FUNCTION_BLOCK FB_TelescopeAuxiliary
VAR
	tempSensorM1   		AT%I*: INT;
	tempSensorM1cell	AT%I*: INT;
	tempSensorM2   		AT%I*: INT;
	tempSensorFlange	AT%I*: INT;
	fbComm				: I_Comm;
END_VAR
VAR_OUTPUT
	tempM1				: REAL;
	tempM1cell			: REAL;
	tempM2				: REAL;
	tempFlange			: REAL;
END_VAR

tempM1 		:= tempSensorM1 / 32767.0 * 150.0 - 50.0; 
tempM1cell 	:= tempSensorM1cell / 32767.0 * 150.0 - 50.0;
tempM2 		:= tempSensorM2 / 32767.0 * 150.0 - 50.0;
tempFlange 	:= tempSensorFlange / 32767.0 * 150.0 - 50.0;

//FB_Init is always available implicitly and it is used primarily for initialization.
//The return value is not evaluated. For a specific influence, you can also declare the
//methods explicitly and provide additional code there with the standard initialization
//code. You can evaluate the return value.
METHOD FB_Init: BOOL
VAR_INPUT
    bInitRetains	: BOOL; // TRUE: the retain variables are initialized (reset warm / reset cold)
    bInCopyCode		: BOOL;  // TRUE: the instance will be copied to the copy code afterward (online change)
	comm			: I_Comm;	   
END_VAR
THIS^.fbComm := comm;
END_METHOD

METHOD SendTelemetry : BOOL
VAR_INPUT
END_VAR
fbComm.Publish('telescope', 'dome', 'AUXILIARY.SENSOR[1].NAME', 'TEMP_M1');
fbComm.Publish('telescope', 'dome', 'AUXILIARY.SENSOR[1].VALUE', LREAL_TO_FMTSTR(tempM1, 2, TRUE));
fbComm.Publish('telescope', 'dome', 'AUXILIARY.SENSOR[1].UNIT', 'C');
fbComm.Publish('telescope', 'dome', 'AUXILIARY.SENSOR[2].NAME', 'TEMP_M2');
fbComm.Publish('telescope', 'dome', 'AUXILIARY.SENSOR[2].VALUE', LREAL_TO_FMTSTR(tempM2, 2, TRUE));
fbComm.Publish('telescope', 'dome', 'AUXILIARY.SENSOR[2].UNIT', 'C');
END_METHOD

END_FUNCTION_BLOCK

(* stored: Version 1.1.0.1, ProductVersion 3.1.4024.15
   POU FB_TelescopeAuxiliary: Id {cb121caa-cba6-4e85-8680-87ba92407bb5}, SpecialFunc None
   Method FB_Init: Id {0ab38d83-c759-49b4-b051-261f5cd152ad}
   Method SendTelemetry: Id {5ed8a466-d7bf-44d5-b9d6-ae006c1229a8} *)
